// TIA Portal V16 export
// export: Created 2024-12-03T15:41:43.175405Z, ExportSetting WithDefaults, DisplayName Totally Integrated Automation Portal, DisplayVersion V16 Update 6, DisplayName TIA Portal Version Control Interface, DisplayVersion V16 Update 2, DisplayName TIA Portal Openness, DisplayVersion V16 Update 6, DisplayName TIA Portal Teamcenter Gateway, DisplayVersion V16, DisplayName SINAMICS Startdrive Advanced, DisplayVersion V16 Update 5, DisplayName SINAMICS Startdrive G130, G150, S120, S150, SINAMICS MV, S210, DisplayVersion V16 Update 5, DisplayName SINAMICS Startdrive G110M, G120, G120C, G120D, G120P, G115D, DisplayVersion V16 Update 5, DisplayName STEP 7 Professional, DisplayVersion V16 Update 6, DisplayName STEP 7 Safety, DisplayVersion V16, DisplayName WinCC Advanced / Unified PC, DisplayVersion V16 Update 6
FUNCTION_BLOCK "ZPA_TransferUnit_Controller"   // FB63, SCL
{ S7_Optimized_Access := 'TRUE' }
VERSION : 0.1
// stored: AutoNumber true, IsIECCheckEnabled false, IsRetainMemResEnabled false, MemoryReserve 100, SetENOAutomatically false, UDAEnableTagReadback false
   VAR_INPUT
      I_BuildName : Bool := true;
      I_ReceivePosition : Int;
      I_SendingPosition : Int;
      I_NoEndSensor : Bool;
      I_SentAtEnd : Bool;
      I_ConnectUpstream : Bool := TRUE;
      I_UpstreamConveyor : "Conveyor_UDT";
      I_DownStreamConveyor : "Conveyor_UDT";
      I_AlignAfterReceive : Bool;
      I_AlignSpeed : Real;
      I_AlignDirection : Bool;
      I_AlignDistance : Real;
      I_AlignPostition : Int;
      I_AlignConveyorIndex : Int;   // 1= recieve / 2 = sending
   END_VAR
   VAR_IN_OUT
      IO_ReceiveConveyor : "Conveyor_UDT";
      IO_SendingConveyor : "Conveyor_UDT";
      IO_VLV_Transfer : "TransferUnitUpDown";
   END_VAR
   VAR
      cycleRun : "CycleRun";
      alarmReceive : "AlarmInfo_UDT";
      alarmSending : "AlarmInfo_UDT";
      StartupDelay { S7_SetPoint := 'True'} : TON_TIME;
      EncoderReceive { S7_SetPoint := 'True'} : "Virtual_Encoder_FB";
      EncoderSending { S7_SetPoint := 'True'} : "Virtual_Encoder_FB";
      DownStreamRunningPredictor { S7_SetPoint := 'True'} : Int;
      DownStreamIsRunning : Bool;
   END_VAR
   VAR RETAIN
      StepNumber : DInt;
      PrevStepNumber : DInt;
   END_VAR
   VAR
      Step_105_GapTimeOk : Bool;
      GapTimeTimer : "TON_Encoder_FB";
      diag : Struct
         TrackingLost : UInt;
      END_STRUCT;
      Step_3110_CHeckConveyorCorrectlyReceived { S7_SetPoint := 'True'} : "StepperController_Encoder";
      Step_31210_CheckCOnveyorCorrectlySent { S7_SetPoint := 'True'} : "StepperController_Encoder";
      Step_Recv_10_WaitingReceive { S7_SetPoint := 'True'} : "StepperController";
      Step_Recv_20_RecevingSingle { S7_SetPoint := 'True'} : "StepperController_Encoder";
      Step_Recv_40_RunEnd { S7_SetPoint := 'True'} : "StepperController_Encoder";
      Step_Recv_50_ReceivePosition { S7_SetPoint := 'True'} : "StepperController_Encoder";
      Step_Recv_55_WaitMotorOff { S7_SetPoint := 'True'} : "StepperController";
      Step_Algign_60 { S7_SetPoint := 'True'} : "StepperController_Encoder";
      Step_Sent_100_RunTillEnd { S7_SetPoint := 'True'} : "StepperController_Encoder";
      Step_Sent_105_RequestSending { S7_SetPoint := 'True'} : "StepperController";
      Step_Sent_110_SentItem { S7_SetPoint := 'True'} : "StepperController_Encoder";
      Step_Sent_120_EmptyRun { S7_SetPoint := 'True'} : "StepperController_Encoder";
      blockedAlarmSending { S7_SetPoint := 'True'} : Program_Alarm;
      blockedAlarmReceiving { S7_SetPoint := 'True'} : Program_Alarm;
   END_VAR
   VAR_TEMP
      T_AppState : "ApplicationState_UDT";
      T_ZoneInfo : "ZoneInfo";
      T_TransferInReceivePosition : Bool;
      T_TransferInSendingPosition : Bool;
      T_Condition : Bool;
      T_NextStep : DInt;
      T_DeltaDistance : Real;
   END_VAR
   VAR CONSTANT
      STEP_60_ALIGNMENT : DInt := 60;
      InitStep : DInt := 3100;
      AlarmReceiveErrorStep : DInt := 910;
      AlarmSendingErrorStep : DInt := 930;
   END_VAR
BEGIN
   #T_ZoneInfo := "ApplicationState_DB".ZoneNames[#IO_SendingConveyor.Zone];
   #T_AppState := "ApplicationState_DB".Appstate[#T_ZoneInfo.AppStateIndex];

   IF #IO_SendingConveyor.Zone <> 0 THEN
       #IO_VLV_Transfer.Zone := #IO_SendingConveyor.Zone;
   END_IF;

   IF "RunTime_DB".CycleRun = #T_ZoneInfo.AppStateIndex THEN
       #cycleRun();
   END_IF;

   REGION COMBINE TRACKING COMMANDS //new tracking only arrives at receive conveyor
       #IO_ReceiveConveyor.TrackingCmd.InductNewTracking := #IO_ReceiveConveyor.TrackingCmd.InductNewTracking
       OR #IO_SendingConveyor.TrackingCmd.InductNewTracking;
       #IO_ReceiveConveyor.TrackingCmd.ClearTracking := #IO_ReceiveConveyor.TrackingCmd.ClearTracking
       OR #IO_SendingConveyor.TrackingCmd.ClearTracking;
   END_REGION

   REGION Receive sent position

       #T_TransferInReceivePosition := #IO_VLV_Transfer.Status.Position = #I_ReceivePosition;
       #T_TransferInSendingPosition := #IO_VLV_Transfer.Status.Position = #I_SendingPosition;

   END_REGION

   REGION ACCUMULATION SENDING

       #IO_SendingConveyor.Status.AccumulationOn :=
       #IO_SendingConveyor.Cmd.Accumulate.Acc_ext_1 OR
       #IO_SendingConveyor.Cmd.Accumulate.Acc_ext_2 OR
       #IO_SendingConveyor.Cmd.Accumulate.Acc_ext_3 OR
       #IO_SendingConveyor.Cmd.Accumulate.Acc_ext_4 OR
       #IO_SendingConveyor.Cmd.Accumulate.Acc_ext_5 OR
       #IO_SendingConveyor.Cmd.Accumulate.Acc_Scale_1 OR
       #IO_SendingConveyor.Cmd.Accumulate.Acc_Scale_2 OR
       #IO_SendingConveyor.Cmd.Accumulate.Acc_Scale_3 OR
       #IO_SendingConveyor.Cmd.Accumulate.Acc_Scan_1 OR
       #IO_SendingConveyor.Cmd.Accumulate.Acc_Scan_2 OR
       #IO_SendingConveyor.Cmd.Accumulate.Acc_Scan_3 OR
       #IO_SendingConveyor.Cmd.Accumulate.Acc_TC_1 OR
       #IO_SendingConveyor.Cmd.Accumulate.Acc_TC_1 OR
       #IO_SendingConveyor.Cmd.Accumulate.Acc_TC_3;

   END_REGION

   REGION Auto MODe

       #IO_SendingConveyor.Status.ReadyForStandby := #StepNumber = 105 OR #StepNumber = 10 OR #StepNumber >= 3110;
       #IO_ReceiveConveyor.Status.ReadyForStandby := #IO_SendingConveyor.Status.ReadyForStandby;

       IF NOT #T_AppState.States.AutoModeActivated.State AND #StepNumber <> 0 THEN
           #PrevStepNumber := #StepNumber;
           #StepNumber := 0;
           #IO_ReceiveConveyor.Status.Initialized := false;
           #IO_SendingConveyor.Status.Initialized := false;
       END_IF;

       IF #T_AppState.States.AutoModeActivated.State AND #StepNumber = 0 THEN
           #StepNumber := #PrevStepNumber;
           //#StepNumber := #InitStep;
       END_IF;

       IF #StepNumber > 0 AND #StepNumber < 3000 THEN
           #IO_ReceiveConveyor.Status.Initialized := TRUE;
           #IO_SendingConveyor.Status.Initialized := TRUE;
           #IO_ReceiveConveyor.Status.StartedAutoMode := TRUE;
           #IO_SendingConveyor.Status.StartedAutoMode := TRUE;
       END_IF;

   END_REGION

   REGION Init steps

       IF #StepNumber = 0 THEN
           #StepNumber := #InitStep;
           #StepNumber := 10;
       END_IF;

       IF #IO_ReceiveConveyor.Cmd.ReInitialize OR #IO_SendingConveyor.Cmd.ReInitialize THEN
           #StepNumber := 0;
           #IO_ReceiveConveyor.Status.Initialized := FALSE;
           #IO_SendingConveyor.Status.Initialized := FALSE;
           #StepNumber := 10;
       END_IF;

       IF #StepNumber = #InitStep AND #IO_SendingConveyor.Input.SensorAtEndLogic.State THEN
           #StepNumber := 100;
       END_IF;

       IF #StepNumber = #InitStep AND (#IO_ReceiveConveyor.Input.SensorAtEndLogic.State AND NOT #I_NoEndSensor) THEN
           #StepNumber := 100;
       END_IF;

       IF #StepNumber = #InitStep THEN
           #StepNumber := 3110;
       END_IF;

       //CHeck if we need to receive an object
       #Step_3110_CHeckConveyorCorrectlyReceived(I_StepNumber := 3110,
                                                 I_NextStepNumber := 100,
                                                 I_TimeOutStepNumber := 3120,
                                                 I_AccumulateConditionTIme := TRUE,
                                                 I_Condition := #IO_ReceiveConveyor.Input.SensorAtEndLogic.State AND NOT #I_NoEndSensor,
                                                 I_PauseTimeOut := NOT #IO_ReceiveConveyor.Input.Running_FB,
                                                 I_TimeOutDistance := #IO_ReceiveConveyor.Settings.Timings.InitDistance,
                                                 I_DeltaDistance := #IO_ReceiveConveyor.Encoder.Distance_mm,
                                                 I_IgnoreTimeOut := FALSE,
                                                 IO_PrevStepNumber := #PrevStepNumber,
                                                 IO_StepNumber := #StepNumber);

       //CHeck if we need to send an object
       #Step_31210_CheckCOnveyorCorrectlySent(I_StepNumber := 3120,
                                              I_NextStepNumber := 100,
                                              I_TimeOutStepNumber := 10,
                                              I_AccumulateConditionTIme := TRUE,
                                              I_Condition := #IO_SendingConveyor.Input.SensorAtEndLogic.State,
                                              I_PauseTimeOut := NOT #IO_SendingConveyor.Input.Running_FB,
                                              I_TimeOutDistance := #IO_SendingConveyor.Settings.Timings.InitDistance,
                                              I_DeltaDistance := #IO_SendingConveyor.Encoder.Distance_mm,
                                              I_IgnoreTimeOut := FALSE,
                                              IO_PrevStepNumber := #PrevStepNumber,
                                              IO_StepNumber := #StepNumber);

   END_REGION

   REGION DOWNSTREAM RUNNING SIMULATOR

       IF #DownStreamRunningPredictor <= 3 THEN
           #DownStreamRunningPredictor += 1;
       END_IF;

       IF NOT #I_DownStreamConveyor.Input.Running_FB THEN
           #DownStreamIsRunning := false;
       END_IF;

       IF #DownStreamRunningPredictor > 3 THEN
           #DownStreamIsRunning := FALSE;
       END_IF;

       IF #Step_Sent_100_RunTillEnd.O_ConditionTrans OR #Step_Sent_110_SentItem.O_ConditionTrans OR #I_DownStreamConveyor.Input.Running_FB THEN
           #DownStreamRunningPredictor := 0;
       END_IF;

       IF #I_DownStreamConveyor.Input.Running_FB OR #DownStreamRunningPredictor < 3 THEN
           #DownStreamIsRunning := true;
       END_IF;


   END_REGION

   REGION Receive conveyor steps

       REGION STEP 10 WAIT TO RECEIVE

           #T_Condition := #I_UpstreamConveyor.Cmd.ReadyToSent AND #I_ConnectUpstream
           AND #T_TransferInReceivePosition;


           #Step_Recv_10_WaitingReceive(I_StepNumber := 10,
                                        I_NextStepNumber := 20,
                                        I_Condition := #T_Condition,
                                        I_IgnoreTimeOut := TRUE,
                                        IO_PrevStepNumber := #PrevStepNumber,
                                        IO_StepNumber := #StepNumber);

       END_REGION

       REGION STEP 20 RECEIVE A SINGLE OBJECT

           #Step_Recv_20_RecevingSingle(I_StepNumber := 20,
                                        I_NextStepNumber := 40,
                                        I_Condition := #IO_ReceiveConveyor.Input.SensorAtStartLogic.FE OR #IO_ReceiveConveyor.Input.SensorAtEndLogic.State,
                                        I_TimeOutStepNumber := 10,
                                        I_DeltaDistance := #IO_ReceiveConveyor.Encoder.Distance_mm,
                                        I_TimeOutDistance := #IO_ReceiveConveyor.Settings.Timings.ConveyorLength,
                                        I_IgnoreTimeOut := FALSE,
                                        IO_PrevStepNumber := #PrevStepNumber,
                                        IO_StepNumber := #StepNumber);

           REGION TRACK RECEIVING HANDLEING

               #IO_ReceiveConveyor.TrackingStat.TrackingReceived := FALSE;
               #IO_ReceiveConveyor.Status.ObjectReceivePulse := FALSE;
               IF #Step_Recv_20_RecevingSingle.O_ConditionTrans AND NOT #IO_ReceiveConveyor.TrackingCmd.InductNewTracking THEN
                   #IO_ReceiveConveyor.TrackingStat.Current := #I_UpstreamConveyor.TrackingStat.InSending;
                   #IO_ReceiveConveyor.TrackingStat.TrackingReceived := TRUE;
                   #IO_ReceiveConveyor.Status.ObjectReceivePulse := TRUE;

                   // //Tracking diagnostics
                   // IF #IO_ReceiveConveyor.TrackingStat.Current.Barcode = '' OR #IO_ReceiveConveyor.TrackingStat.Current.PLC_Dest = 0 THEN
                   //     #IO_ReceiveConveyor.TrackingStat.Current.Barcode := 'TRACKING_LOST';
                   //     #IO_ReceiveConveyor.TrackingStat.Current.PLC_Dest := 99;
                   //     #diag.TrackingLost += 1;
                   // END_IF;

               END_IF;

               IF #Step_Recv_20_RecevingSingle.O_ConditionTrans AND #IO_ReceiveConveyor.TrackingCmd.InductNewTracking THEN
                   #IO_ReceiveConveyor.TrackingStat.Current := #IO_ReceiveConveyor.TrackingCmd.NewTrackingId;
                   #IO_ReceiveConveyor.TrackingCmd.InductNewTracking := FALSE;
                   #IO_ReceiveConveyor.TrackingStat.TrackingReceived := TRUE;
               END_IF;

           END_REGION

       END_REGION

       REGION STEP 40 RUN THE OBJECT TILL THE END AT RECEIVING

           IF #I_NoEndSensor THEN
               #T_Condition := #IO_ReceiveConveyor.Input.SensorAtStartLogic.FE;
           ELSE
               #T_Condition := #IO_ReceiveConveyor.Input.SensorAtEndLogic.State;
           END_IF;

           #Step_Recv_40_RunEnd(I_StepNumber := 40,
                                I_NextStepNumber := 50,
                                I_TimeOutStepNumber := #AlarmReceiveErrorStep,
                                I_Condition := #T_Condition,
                                I_IgnoreTimeOut := FALSE,
                                I_DeltaDistance := #IO_ReceiveConveyor.Encoder.Distance_mm,
                                I_TimeOutDistance := #IO_ReceiveConveyor.Settings.Timings.ConveyorLength,
                                IO_PrevStepNumber := #PrevStepNumber,
                                IO_StepNumber := #StepNumber);

       END_REGION

       REGION STEP 50 POSITION THE OBJECT

           #Step_Recv_50_ReceivePosition(I_StepNumber := 50,
                                         I_NextStepNumber := 55,
                                         I_Condition := #IO_ReceiveConveyor.Input.Running_FB,
                                         I_DeltaDistance := #IO_ReceiveConveyor.Encoder.Distance_mm,
                                         I_ConditionDistance := #IO_ReceiveConveyor.Settings.Timings.ReceiveDistance,
                                         I_AccumulateConditionTIme := TRUE,
                                         I_IgnoreTimeOut := TRUE,
                                         IO_PrevStepNumber := #PrevStepNumber,
                                         IO_StepNumber := #StepNumber);

       END_REGION

       REGION STEP 55 WAIT UNTILL MOTOR IS STOPPED

           IF #I_AlignAfterReceive THEN
               #T_NextStep := #STEP_60_ALIGNMENT;
           ELSE
               #T_NextStep := 100;
           END_IF;

           #Step_Recv_55_WaitMotorOff(I_StepNumber := 55,
                                      I_NextStepNumber := #T_NextStep,
                                      I_Condition := NOT #IO_ReceiveConveyor.Input.Running_FB,
                                      I_ConditionTIme := #IO_SendingConveyor.Settings.Timings.DelayedStart,
                                      I_AccumulateConditionTIme := TRUE,
                                      I_IgnoreTimeOut := TRUE,
                                      IO_PrevStepNumber := #PrevStepNumber,
                                      IO_StepNumber := #StepNumber);

       END_REGION

   END_REGION

   REGION ALIGNMENT

       REGION STEP 60 ALIGNEMENT

           IF #I_AlignConveyorIndex = 1 THEN
               #T_Condition := #IO_ReceiveConveyor.Input.Running_FB;
               #T_DeltaDistance := #IO_ReceiveConveyor.Encoder.Distance_mm;
           ELSIF #I_AlignConveyorIndex = 2 THEN
               #T_Condition := #IO_SendingConveyor.Input.Running_FB;
               #T_DeltaDistance := #IO_SendingConveyor.Encoder.Distance_mm;
           END_IF;

           #Step_Algign_60(I_StepNumber:=#STEP_60_ALIGNMENT,
                           I_NextStepNumber:=100,
                           I_Condition:=#T_Condition,
                           I_ConditionDistance:=#I_AlignDistance,
                           I_DeltaDistance:=#T_DeltaDistance,
                           I_IgnoreTimeOut:=TRUE,
                           IO_StepNumber:=#StepNumber,
                           IO_PrevStepNumber:=#PrevStepNumber);

       END_REGION


   END_REGION

   REGION Sending conveyor steps

       IF #I_SentAtEnd
           AND #IO_SendingConveyor.Input.SensorAtEndLogic.State
           AND NOT #IO_ReceiveConveyor.Cmd.RunAuto
           AND #StepNumber = 10 THEN
           #StepNumber := 100;
       END_IF;

       REGION STEP 100 WAIT TO SENT
           #Step_Sent_100_RunTillEnd(I_StepNumber := 100,
                                     I_NextStepNumber := 105,
                                     I_TimeOutStepNumber := #AlarmSendingErrorStep,
                                     I_Condition := (#IO_SendingConveyor.Input.SensorAtEndLogic.State
                                     AND #T_TransferInSendingPosition)
                                     AND NOT #T_AppState.States.RequestingAutoModeOff
                                     AND NOT #T_AppState.States.Standby.State,
                                     I_IgnoreTimeOut := #IO_SendingConveyor.Input.SensorAtEndLogic.State OR NOT #IO_SendingConveyor.Input.Running_FB,
                                     I_DeltaDistance := #IO_SendingConveyor.Encoder.Distance_mm,
                                     I_TimeOutDistance := #IO_SendingConveyor.Settings.Timings.ConveyorLength,
                                     IO_PrevStepNumber := #PrevStepNumber,
                                     IO_StepNumber := #StepNumber);

           IF #Step_Sent_100_RunTillEnd.O_ConditionTrans THEN
               #IO_ReceiveConveyor.TrackingStat.InSending := #IO_ReceiveConveyor.TrackingStat.Current;
               #IO_SendingConveyor.TrackingStat.InSending := #IO_ReceiveConveyor.TrackingStat.Current;
           END_IF;

       END_REGION

       REGION STEP 105 CHECK DOWNSTREAM IS READY

           REGION GAP TIME OK

               #GapTimeTimer(I_DeltaDistance_mm := #I_DownStreamConveyor.Encoder.Distance_mm,
                             I_SetPoint := #IO_SendingConveyor.Settings.Timings.GapDistance,
                             I_Start := #I_DownStreamConveyor.Input.Running_FB,
                             I_Remanent := TRUE,
                             I_Reset := #IO_SendingConveyor.Input.SensorAtEndLogic.FE,
                             Q => #Step_105_GapTimeOk);

               IF #IO_SendingConveyor.Settings.Timings.GapDistance = 0.0 THEN
                   #Step_105_GapTimeOk := true;
               END_IF;

           END_REGION

           #Step_Sent_105_RequestSending(I_StepNumber := 105,
                                         I_NextStepNumber := 110,
                                         I_Condition := #I_DownStreamConveyor.Cmd.ReadyToReceive AND #T_TransferInSendingPosition
                                         AND #IO_SendingConveyor.Input.SensorAtEndLogic.State AND #Step_105_GapTimeOk
                                         AND NOT #IO_SendingConveyor.Status.AccumulationOn,
                                         I_IgnoreTimeOut := TRUE,
                                         I_PauseTimeOut := NOT #IO_SendingConveyor.Input.Running_FB,
                                         IO_PrevStepNumber := #PrevStepNumber,
                                         IO_StepNumber := #StepNumber);
       END_REGION

       REGION STEP 110 SENT OBJECT
           #Step_Sent_110_SentItem(I_StepNumber := 110,
                                   I_NextStepNumber := 120,
                                   I_TimeOutStepNumber := #AlarmSendingErrorStep,
                                   I_Condition := NOT #IO_SendingConveyor.Input.SensorAtEndLogic.State,
                                   I_DeltaDistance := #IO_SendingConveyor.Encoder.Distance_mm,
                                   I_TimeOutDistance := #IO_SendingConveyor.Settings.Timings.ConveyorLength,
                                   I_IgnoreTimeOut := FALSE,
                                   I_PauseTimeOut := NOT #IO_SendingConveyor.Input.Running_FB,
                                   IO_PrevStepNumber := #PrevStepNumber,
                                   IO_StepNumber := #StepNumber);

           #IO_SendingConveyor.Status.ObjectSentPulse := #Step_Sent_110_SentItem.O_ConditionTrans;

       END_REGION

       REGION STEP 120 RUN EMPTY (RUN WITH SENDING HOLD ON TIME)
           #Step_Sent_120_EmptyRun(I_StepNumber := 120,
                                   I_NextStepNumber := 10,
                                   I_Condition := NOT #IO_SendingConveyor.Input.SensorAtEndLogic.State AND #IO_SendingConveyor.Input.Running_FB,
                                   I_DeltaDistance := #IO_SendingConveyor.Encoder.Distance_mm,
                                   I_ConditionDistance := #IO_SendingConveyor.Settings.Timings.SendDistance,
                                   I_IgnoreTimeOut := TRUE,
                                   IO_PrevStepNumber := #PrevStepNumber,
                                   IO_StepNumber := #StepNumber);
       END_REGION

   END_REGION

   REGION Reset stepnumber AND status when object is removed AND conveyor was NOT running

       IF #IO_SendingConveyor.Input.SensorAtEndLogic.FE
           AND #StepNumber <> 120
           AND NOT #IO_SendingConveyor.Cmd.RunAuto THEN
           // #IO_COnv.TrackingCmd.ClearTracking := TRUE;
           #StepNumber := 10;
           //#StepNumber := 8000;
       END_IF;

   END_REGION

   REGION STATUS

       #IO_ReceiveConveyor.Status.ExecutingReceiveSequence := #StepNumber > 10 AND #StepNumber <= 55;
       #IO_SendingConveyor.Status.ExecutingSendingSequence := #StepNumber >= 100 AND #StepNumber <= 120;

       #IO_SendingConveyor.Status.RequestForSending := #StepNumber = 40 OR #StepNumber = 50 OR
       #StepNumber = 100 OR
       #StepNumber = 105 OR #StepNumber = 110;


       #IO_ReceiveConveyor.Status.ObjectOnConveyor := #StepNumber > 20 AND #StepNumber < 120;

       #IO_ReceiveConveyor.Status.Empty := #StepNumber = 10 OR #StepNumber = 20;
       #IO_SendingConveyor.Status.Empty := #StepNumber = 10 OR #StepNumber = 20;

   END_REGION

   REGION Command transfer unit

       IF #IO_ReceiveConveyor.Status.ExecutingReceiveSequence
           OR #StepNumber = 10
           OR #StepNumber = 3110
       THEN
           #IO_VLV_Transfer.Cmd.InAuto := #I_ReceivePosition = "Down";
       END_IF;


       IF #IO_SendingConveyor.Status.ExecutingSendingSequence
           OR #StepNumber = 3120
       THEN
           #IO_VLV_Transfer.Cmd.InAuto := #I_SendingPosition = "Down";
       END_IF;

       IF #StepNumber = #STEP_60_ALIGNMENT THEN
           #IO_VLV_Transfer.Cmd.InAuto := #I_AlignPostition = "Down";
       END_IF;

   END_REGION

   REGION CLEAR TRACKING

       IF #I_DownStreamConveyor.TrackingStat.TrackingReceived OR #IO_ReceiveConveyor.TrackingCmd.ClearTracking THEN
           //#IO_ReceiveConveyor.TrackingStat.Current := "Tracking_DB".EmptyTrackingSimple;
           #IO_ReceiveConveyor.TrackingStat.InSending := "Tracking_DB".EmptyTrackingSimple;
           #IO_ReceiveConveyor.TrackingCmd.ClearTracking := FALSE;
       END_IF;

   END_REGION

   REGION TRANSFER TRACKING BETWEEN INTERNAL SENDING AND RECEIVING

       #IO_SendingConveyor.TrackingCmd := #IO_ReceiveConveyor.TrackingCmd;
       #IO_SendingConveyor.TrackingStat := #IO_ReceiveConveyor.TrackingStat;

   END_REGION

   REGION Interfacing receive conveyor

       #IO_ReceiveConveyor.Cmd.ReadyToReceive := #StepNumber = 10 OR #StepNumber = 20 OR #StepNumber = 40 OR #StepNumber = 50;
       #IO_ReceiveConveyor.Cmd.ReadyToReceive := #IO_ReceiveConveyor.Cmd.ReadyToReceive AND #T_TransferInReceivePosition;
       #IO_ReceiveConveyor.Cmd.RunAuto := #StepNumber = 20 OR #StepNumber = 40 OR #StepNumber = 50 OR #StepNumber = 3110;

       #IO_ReceiveConveyor.Cmd.RunAuto := #IO_ReceiveConveyor.Cmd.RunAuto OR (#StepNumber = #STEP_60_ALIGNMENT AND #I_AlignConveyorIndex = 1);

       #IO_ReceiveConveyor.Cmd.RunAuto := #IO_ReceiveConveyor.Cmd.RunAuto AND #T_TransferInReceivePosition;

   END_REGION

   REGION Interfacing sending conveyor

       #IO_SendingConveyor.Cmd.ReadyToSent := (#StepNumber = 105 AND NOT #IO_SendingConveyor.Status.AccumulationOn) OR #StepNumber = 110;
       #IO_SendingConveyor.Cmd.ReadyToSent := #IO_SendingConveyor.Cmd.ReadyToSent AND #T_TransferInSendingPosition;

       #IO_SendingConveyor.Cmd.RunAuto :=  #StepNumber = 105 OR #StepNumber = 110 OR #StepNumber = 120;
       #IO_SendingConveyor.Cmd.RunAuto := #IO_SendingConveyor.Cmd.RunAuto AND (#DownStreamIsRunning OR #StepNumber = 120);

       #IO_SendingConveyor.Cmd.RunAuto := #IO_SendingConveyor.Cmd.RunAuto AND (#I_DownStreamConveyor.Cmd.ReadyToReceive OR #StepNumber = 120);
       #IO_SendingConveyor.Cmd.RunAuto := #IO_SendingConveyor.Cmd.RunAuto OR #StepNumber = 3120;
       #IO_SendingConveyor.Cmd.RunAuto := #IO_SendingConveyor.Cmd.RunAuto OR (#StepNumber = 100 AND NOT #T_AppState.States.Standby.State);

       #IO_SendingConveyor.Cmd.RunAuto := #IO_SendingConveyor.Cmd.RunAuto OR (#StepNumber = #STEP_60_ALIGNMENT AND #I_AlignConveyorIndex = 2);

       #IO_SendingConveyor.Cmd.RunAuto := #IO_SendingConveyor.Cmd.RunAuto AND #T_TransferInSendingPosition;

   END_REGION

   REGION DIRECTION

       IF #StepNumber = #STEP_60_ALIGNMENT THEN
           IF #I_AlignDirection THEN
               IF #I_AlignConveyorIndex = 1 THEN
                   #IO_ReceiveConveyor.Cmd.Direction := NOT #IO_ReceiveConveyor.Cmd.Direction;
               ELSIF #I_AlignConveyorIndex = 1 THEN
                   #IO_SendingConveyor.Cmd.Direction := NOT #IO_SendingConveyor.Cmd.Direction;
               END_IF;
           END_IF;
       END_IF;

   END_REGION

   REGION Speed controller

       #IO_ReceiveConveyor.Cmd.SpeedAuto := #IO_ReceiveConveyor.Settings.Speed.speed;

       IF #IO_ReceiveConveyor.Settings.Speed.speedController AND #I_ConnectUpstream THEN
           IF #IO_ReceiveConveyor.Input.SensorAtStartLogic.State THEN
               #IO_ReceiveConveyor.Cmd.SpeedAuto := #I_UpstreamConveyor.Cmd.SpeedAuto * #IO_ReceiveConveyor.Settings.Speed.UpstreamGain;
           END_IF;
       END_IF;

       #IO_SendingConveyor.Cmd.SpeedAuto := #IO_SendingConveyor.Settings.Speed.speed;

       REGION SPEED FOR ALIGNMENT
           IF #StepNumber = #STEP_60_ALIGNMENT THEN
               IF #I_AlignConveyorIndex = 1 THEN
                   #IO_ReceiveConveyor.Cmd.SpeedAuto := #I_AlignSpeed;
               ELSIF #I_AlignConveyorIndex = 2 THEN
                   #IO_SendingConveyor.Cmd.SpeedAuto := #I_AlignSpeed;
               END_IF;
           END_IF;
       END_REGION

   END_REGION

   REGION ALARMS

       REGION Alarms receive conveyor

           #IO_SendingConveyor.Alarms.BlockedReceive.Active :=
           #IO_ReceiveConveyor.Alarms.BlockedReceive.Active := 0;

           #IO_ReceiveConveyor.Alarms.BlockedReceive.Active :=
           #IO_SendingConveyor.Alarms.Status.%X0 :=
           #IO_ReceiveConveyor.Alarms.Status.%X0 := #StepNumber = #AlarmReceiveErrorStep;

           IF #IO_ReceiveConveyor.Alarms.Status > 0 THEN
               "ApplicationState_DB".Appstate[#T_ZoneInfo.AppStateIndex].Alarms.AlarmActiveInternalPLC := TRUE;
           END_IF;

           IF #cycleRun.O_Cycle = 8 THEN

               IF #I_BuildName AND (#IO_ReceiveConveyor.Name = '' OR "HMI_DB".ReloadSettings.signal) THEN
                   #IO_ReceiveConveyor.Name := "buildObjectName"(I_Symbolname := GetSymbolName(variable := #IO_ReceiveConveyor, size := 100));
                   #alarmReceive.info := "buildAlarmInfo"(I_ObjectName := #IO_ReceiveConveyor.Name,
                                                          I_ZoneIndex := #IO_ReceiveConveyor.Zone, I_ZoneName := #T_ZoneInfo.ZoneName);
               END_IF;
               #blockedAlarmReceiving(SIG := #IO_ReceiveConveyor.Alarms.BlockedReceive.Active,
                                      SD_1 := #T_ZoneInfo.ZoneName,
                                      SD_2 := #IO_ReceiveConveyor.Name,
                                      SD_3 := #alarmReceive.info);
           END_IF;

       END_REGION

       REGION Alarms sending conveyor

           #IO_SendingConveyor.Alarms.BlockedSending.Active :=
           #IO_ReceiveConveyor.Alarms.BlockedSending.Active := 0;

           #IO_SendingConveyor.Alarms.BlockedSending.Active :=
           #IO_ReceiveConveyor.Alarms.Status.%X1 :=
           #IO_SendingConveyor.Alarms.Status.%X1 := #StepNumber = #AlarmSendingErrorStep;

           IF #IO_SendingConveyor.Alarms.Status > 0 THEN
               "ApplicationState_DB".Appstate[#T_ZoneInfo.AppStateIndex].Alarms.AlarmActiveInternalPLC := TRUE;
           END_IF;

           IF #cycleRun.O_Cycle = 10 THEN
               IF #I_BuildName AND (#IO_SendingConveyor.Name = '' OR "HMI_DB".ReloadSettings.signal) THEN
                   #IO_SendingConveyor.Name := "buildObjectName"(I_Symbolname := GetSymbolName(variable := #IO_SendingConveyor, size := 100));
                   #alarmSending.info := "buildAlarmInfo"(I_ObjectName := #IO_SendingConveyor.Name,
                                                          I_ZoneIndex := #IO_SendingConveyor.Zone, I_ZoneName := #T_ZoneInfo.ZoneName);
               END_IF;

               #blockedAlarmSending(SIG := #IO_SendingConveyor.Alarms.BlockedReceive.Active,
                                    SD_1 := #T_ZoneInfo.ZoneName,
                                    SD_2 := #IO_SendingConveyor.Name,
                                    SD_3 := #alarmSending.info);
           END_IF;
       END_REGION

       REGION RESET ALARMS

           IF (#T_AppState.Hmi_Buttons.reset.state.State
               OR "Inputs_DB".Reset_System.State
               OR #IO_ReceiveConveyor.Cmd.Reset
               OR #IO_SendingConveyor.Cmd.Reset
               OR #IO_ReceiveConveyor.Cmd.ReInitialize
               OR #IO_SendingConveyor.Cmd.ReInitialize)
               AND (#IO_ReceiveConveyor.Alarms.Status > 0
               OR #IO_SendingConveyor.Alarms.Status > 0)
           THEN
               #IO_ReceiveConveyor.Alarms.BlockedReceive.Active := FALSE;
               #IO_ReceiveConveyor.Alarms.BlockedSending.Active := FALSE;
               #IO_SendingConveyor.Alarms.BlockedSending.Active := FALSE;
               #IO_SendingConveyor.Alarms.BlockedReceive.Active := FALSE;
               #StepNumber := 10;
           END_IF;



       END_REGION

       REGION ACK ALARM
           // IF (#IO_ReceiveConveyor.Alarms.BlockedReceive.Active
           //     OR #IO_SendingConveyor.Alarms.BlockedReceive.Active)
           //     AND #T_AppState.Hmi_Buttons.reset.state.LE THEN
           //     #StepNumber := #PrevStepNumber;
           // END_IF;
       END_REGION

   END_REGION

   REGION AUTO RESET
       IF #IO_SendingConveyor.Alarms.Status > 0
           AND #StepNumber = #AlarmSendingErrorStep
           AND NOT #I_NoEndSensor
           AND NOT #IO_SendingConveyor.Input.Running_FB
           AND #IO_SendingConveyor.Input.SensorAtEndLogic.FE THEN
           #StepNumber := 10;
           #IO_ReceiveConveyor.Alarms := "CONV_DB".empty.Alarms;
           #IO_SendingConveyor.Alarms := "CONV_DB".empty.Alarms;
       END_IF;

       IF #IO_ReceiveConveyor.Alarms.Status > 0
           AND #StepNumber = #AlarmReceiveErrorStep
           AND NOT #I_NoEndSensor
           AND NOT #IO_ReceiveConveyor.Input.Running_FB
           AND #IO_ReceiveConveyor.Input.SensorAtStartLogic.FE THEN
           #IO_ReceiveConveyor.Alarms := "CONV_DB".empty.Alarms;
           #IO_SendingConveyor.Alarms := "CONV_DB".empty.Alarms;
           #StepNumber := 10;
       END_IF;

   END_REGION

   REGION ENCODER RECEIVE

       IF #IO_ReceiveConveyor.Cmd.RunAuto AND #IO_ReceiveConveyor.Input.Running_FB THEN
           #EncoderReceive.I_CurrentRelativeSpeed_Perc := #IO_ReceiveConveyor.Cmd.SpeedAuto;
       ELSE
           #EncoderReceive.I_CurrentRelativeSpeed_Perc := 0.0;
       END_IF;

       #EncoderReceive(I_RelativeReferenceSpeed_Perc := #IO_ReceiveConveyor.Encoder.Settings.BaseRelative,
                       I_AbsoluteSpeedOnReferecne_m_min := #IO_ReceiveConveyor.Encoder.Settings.Base_M_min,
                       IO_VirtualEncoder := #IO_ReceiveConveyor.Encoder);



   END_REGION

   REGION ENCODER SENDING

       IF #IO_SendingConveyor.Cmd.RunAuto AND #IO_SendingConveyor.Input.Running_FB THEN
           #EncoderSending.I_CurrentRelativeSpeed_Perc := #IO_SendingConveyor.Cmd.SpeedAuto;
       ELSE
           #EncoderSending.I_CurrentRelativeSpeed_Perc := 0.0;
       END_IF;

       #EncoderSending(I_RelativeReferenceSpeed_Perc := #IO_SendingConveyor.Encoder.Settings.BaseRelative,
                       I_AbsoluteSpeedOnReferecne_m_min := #IO_SendingConveyor.Encoder.Settings.Base_M_min,
                       IO_VirtualEncoder := #IO_SendingConveyor.Encoder);



   END_REGION

   #IO_ReceiveConveyor.Cmd.Reset := FALSE;
   #IO_SendingConveyor.Cmd.Reset := FALSE;
   #IO_ReceiveConveyor.Cmd.ReInitialize := FALSE;
   #IO_SendingConveyor.Cmd.ReInitialize := FALSE;
END_FUNCTION_BLOCK
